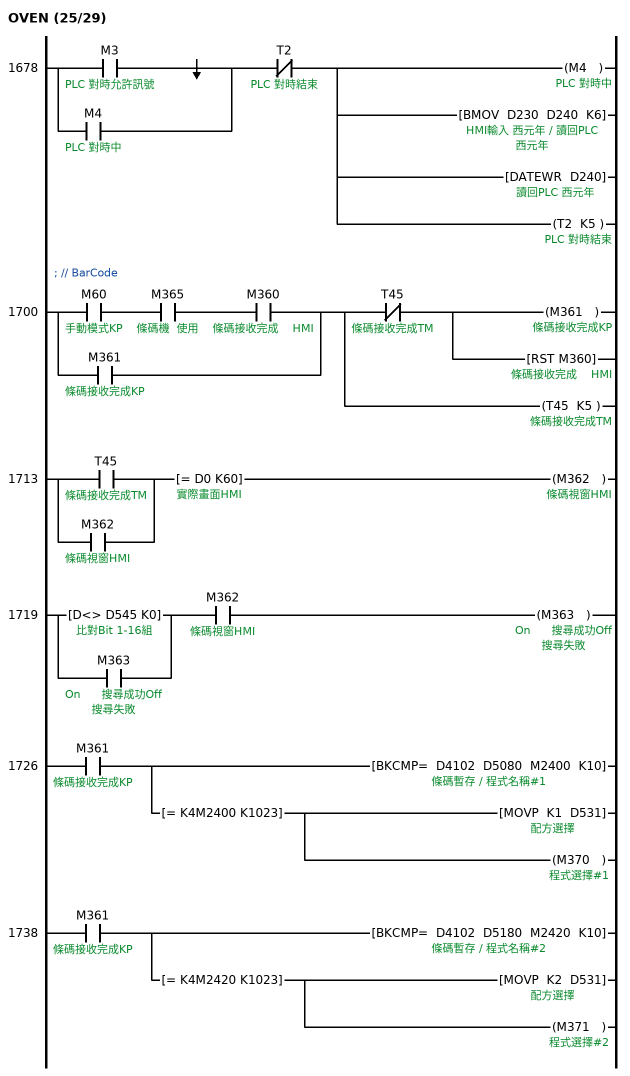
[picture p24: ladder of OVEN, rungs at steps 1678 to 1738]
1678  LD      M3  ; PLC 對時允許訊號
      MEF
      OR      M4  ; PLC 對時中
      ANI     T2  ; PLC 對時結束
      OUT     M4  ; PLC 對時中
      BMOV    D230 D240 K6
      DATEWR  D240
      OUT     T2 K5  ; PLC 對時結束
; // BarCode
1700  LD      M60  ; 手動模式KP
      AND     M365  ; 條碼機  使用
      AND     M360  ; 條碼接收完成    HMI
      OR      M361  ; 條碼接收完成KP
      MPS
      ANI     T45  ; 條碼接收完成TM
      OUT     M361  ; 條碼接收完成KP
      RST     M360  ; 條碼接收完成    HMI
      MPP
      OUT     T45 K5  ; 條碼接收完成TM
1713  LD      T45  ; 條碼接收完成TM
      OR      M362  ; 條碼視窗HMI
      AND=    D0 K60  ; 實際畫面HMI
      OUT     M362  ; 條碼視窗HMI
1719  LDD<>   D545 K0  ; 比對Bit 1-16組
      OR      M363  ; On      搜尋成功Off     搜尋失敗
      AND     M362  ; 條碼視窗HMI
      OUT     M363  ; On      搜尋成功Off     搜尋失敗
1726  LD      M361  ; 條碼接收完成KP
      BKCMP=  D4102 D5080 M2400 K10  ; 條碼暫存 / 程式名稱#1
      AND=    K4M2400 K1023
      MOVP    K1 D531
      OUT     M370  ; 程式選擇#1
1738  LD      M361  ; 條碼接收完成KP
      BKCMP=  D4102 D5180 M2420 K10  ; 程式名稱#2
      AND=    K4M2420 K1023
      MOVP    K2 D531
      OUT     M371  ; 程式選擇#2
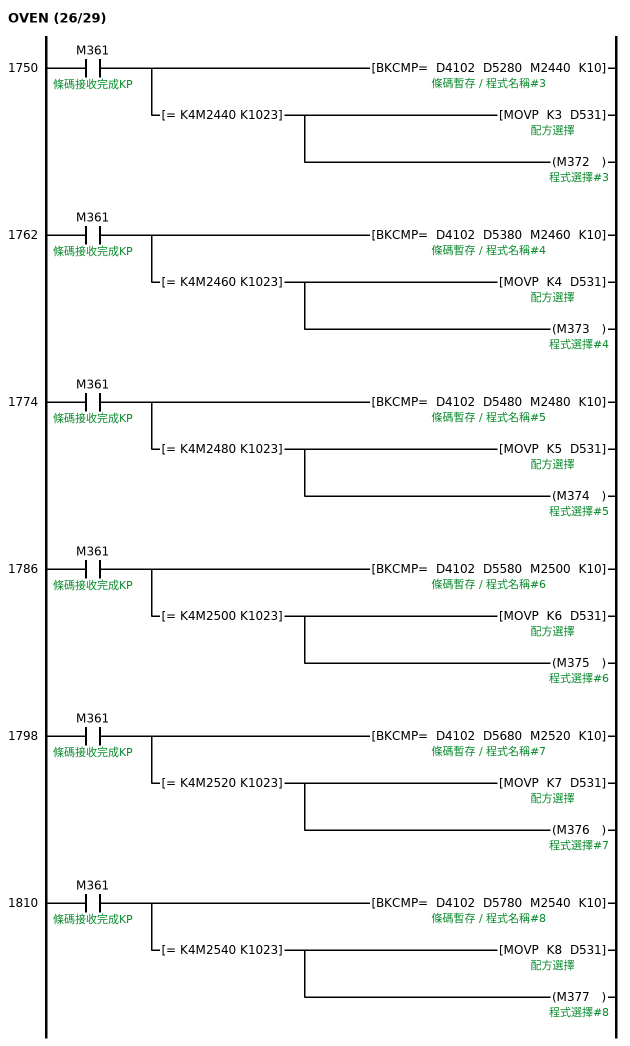
1750  LD      M361  ; 條碼接收完成KP
      BKCMP=  D4102 D5280 M2440 K10  ; 程式名稱#3
      AND=    K4M2440 K1023
      MOVP    K3 D531
      OUT     M372  ; 程式選擇#3
1762  LD      M361  ; 條碼接收完成KP
      BKCMP=  D4102 D5380 M2460 K10  ; 程式名稱#4
      AND=    K4M2460 K1023
      MOVP    K4 D531
      OUT     M373  ; 程式選擇#4
1774  LD      M361  ; 條碼接收完成KP
      BKCMP=  D4102 D5480 M2480 K10  ; 程式名稱#5
      AND=    K4M2480 K1023
      MOVP    K5 D531
      OUT     M374  ; 程式選擇#5
1786  LD      M361  ; 條碼接收完成KP
      BKCMP=  D4102 D5580 M2500 K10  ; 程式名稱#6
      AND=    K4M2500 K1023
      MOVP    K6 D531
      OUT     M375  ; 程式選擇#6
1798  LD      M361  ; 條碼接收完成KP
      BKCMP=  D4102 D5680 M2520 K10  ; 程式名稱#7
      AND=    K4M2520 K1023
      MOVP    K7 D531
      OUT     M376  ; 程式選擇#7
1810  LD      M361  ; 條碼接收完成KP
      BKCMP=  D4102 D5780 M2540 K10  ; 程式名稱#8
      AND=    K4M2540 K1023
      MOVP    K8 D531
      OUT     M377  ; 程式選擇#8
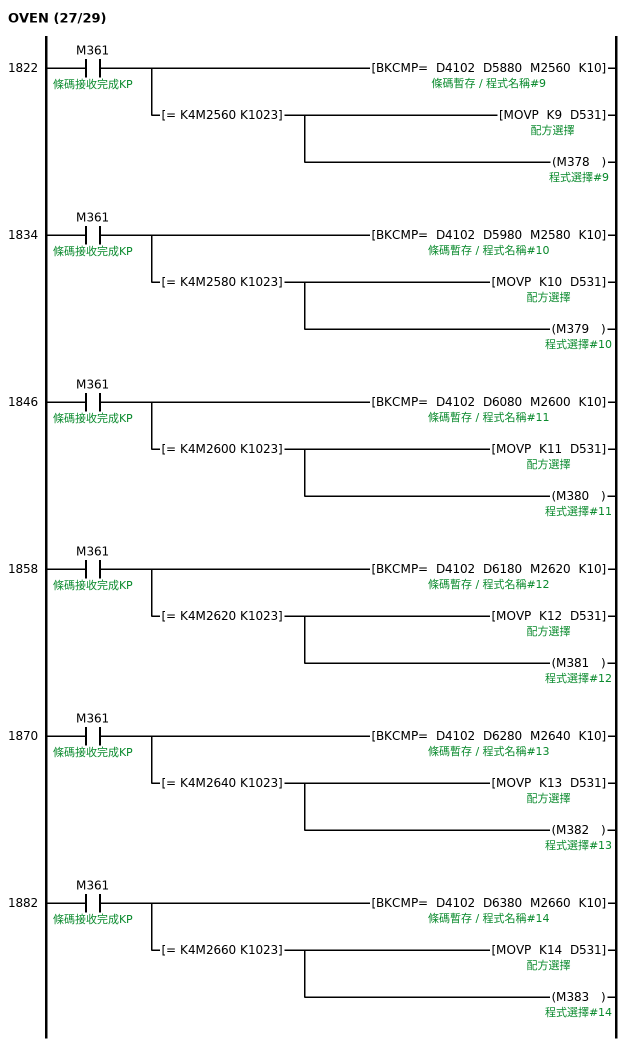
1822  LD      M361  ; 條碼接收完成KP
      BKCMP=  D4102 D5880 M2560 K10  ; 程式名稱#9
      AND=    K4M2560 K1023
      MOVP    K9 D531
      OUT     M378  ; 程式選擇#9
1834  LD      M361  ; 條碼接收完成KP
      BKCMP=  D4102 D5980 M2580 K10  ; 程式名稱#10
      AND=    K4M2580 K1023
      MOVP    K10 D531
      OUT     M379  ; 程式選擇#10
1846  LD      M361  ; 條碼接收完成KP
      BKCMP=  D4102 D6080 M2600 K10  ; 程式名稱#11
      AND=    K4M2600 K1023
      MOVP    K11 D531
      OUT     M380  ; 程式選擇#11
1858  LD      M361  ; 條碼接收完成KP
      BKCMP=  D4102 D6180 M2620 K10  ; 程式名稱#12
      AND=    K4M2620 K1023
      MOVP    K12 D531
      OUT     M381  ; 程式選擇#12
1870  LD      M361  ; 條碼接收完成KP
      BKCMP=  D4102 D6280 M2640 K10  ; 程式名稱#13
      AND=    K4M2640 K1023
      MOVP    K13 D531
      OUT     M382  ; 程式選擇#13
1882  LD      M361  ; 條碼接收完成KP
      BKCMP=  D4102 D6380 M2660 K10  ; 程式名稱#14
      AND=    K4M2660 K1023
      MOVP    K14 D531
      OUT     M383  ; 程式選擇#14
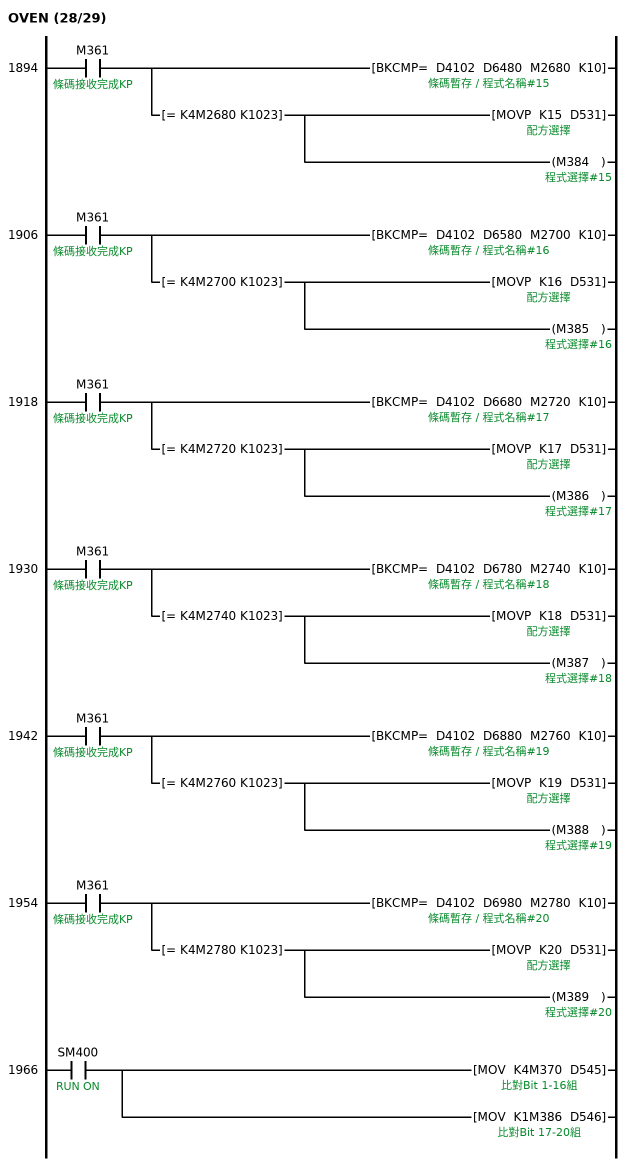
1894  LD      M361  ; 條碼接收完成KP
      BKCMP=  D4102 D6480 M2680 K10  ; 程式名稱#15
      AND=    K4M2680 K1023
      MOVP    K15 D531
      OUT     M384  ; 程式選擇#15
1906  LD      M361  ; 條碼接收完成KP
      BKCMP=  D4102 D6580 M2700 K10  ; 程式名稱#16
      AND=    K4M2700 K1023
      MOVP    K16 D531
      OUT     M385  ; 程式選擇#16
1918  LD      M361  ; 條碼接收完成KP
      BKCMP=  D4102 D6680 M2720 K10  ; 程式名稱#17
      AND=    K4M2720 K1023
      MOVP    K17 D531
      OUT     M386  ; 程式選擇#17
1930  LD      M361  ; 條碼接收完成KP
      BKCMP=  D4102 D6780 M2740 K10  ; 程式名稱#18
      AND=    K4M2740 K1023
      MOVP    K18 D531
      OUT     M387  ; 程式選擇#18
1942  LD      M361  ; 條碼接收完成KP
      BKCMP=  D4102 D6880 M2760 K10  ; 程式名稱#19
      AND=    K4M2760 K1023
      MOVP    K19 D531
      OUT     M388  ; 程式選擇#19
1954  LD      M361  ; 條碼接收完成KP
      BKCMP=  D4102 D6980 M2780 K10  ; 程式名稱#20
      AND=    K4M2780 K1023
      MOVP    K20 D531
      OUT     M389  ; 程式選擇#20
1966  LD      SM400  ; RUN ON
      MOV     K4M370 D545
      MOV     K1M386 D546  ; 比對Bit 17-20組
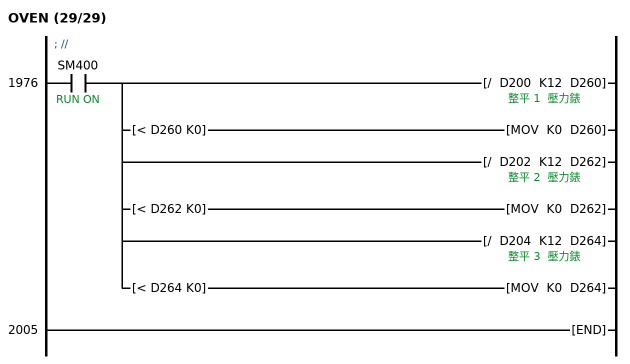
; //
1976  LD      SM400  ; RUN ON
      /       D200 K12 D260  ; 整平 1  壓力錶
      MPS
      AND<    D260 K0
      MOV     K0 D260
      MPP
      /       D202 K12 D262  ; 整平 2  壓力錶
      MPS
      AND<    D262 K0
      MOV     K0 D262
      MPP
      /       D204 K12 D264  ; 整平 3  壓力錶
      AND<    D264 K0
      MOV     K0 D264
2005  END
END_PROGRAM

PROGRAM SECS
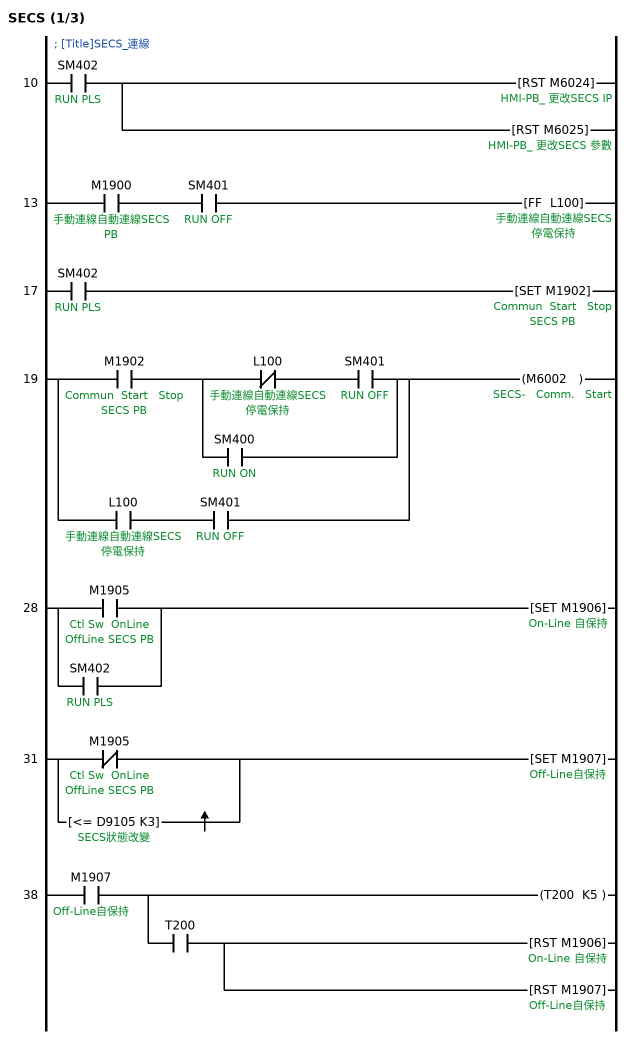
; [Title]SECS_連線
10    LD      SM402  ; RUN PLS
      RST     M6024  ; HMI-PB_ 更改SECS IP
      RST     M6025  ; HMI-PB_ 更改SECS 參數
13    LD      M1900  ; 手動連線自動連線SECS PB
      AND     SM401  ; RUN OFF
      FF      L100  ; 手動連線自動連線SECS    停電保持
17    LD      SM402  ; RUN PLS
      SET     M1902  ; Commun  Start   Stop    SECS PB
19    LD      M1902  ; Commun  Start   Stop    SECS PB
      LDI     L100  ; 手動連線自動連線SECS    停電保持
      AND     SM401  ; RUN OFF
      OR      SM400  ; RUN ON
      ANB
      LD      L100  ; 手動連線自動連線SECS    停電保持
      AND     SM401  ; RUN OFF
      ORB
      OUT     M6002  ; SECS-   Comm.   Start
28    LD      M1905  ; Ctl Sw  OnLine  OffLine SECS PB
      OR      SM402  ; RUN PLS
      SET     M1906  ; On-Line 自保持
31    LDI     M1905  ; Ctl Sw  OnLine  OffLine SECS PB
      LD<=    D9105 K3  ; SECS狀態改變
      MEP
      ORB
      SET     M1907  ; Off-Line自保持
38    LD      M1907  ; Off-Line自保持
      OUT     T200 K5
      AND     T200
      RST     M1906  ; On-Line 自保持
      RST     M1907  ; Off-Line自保持
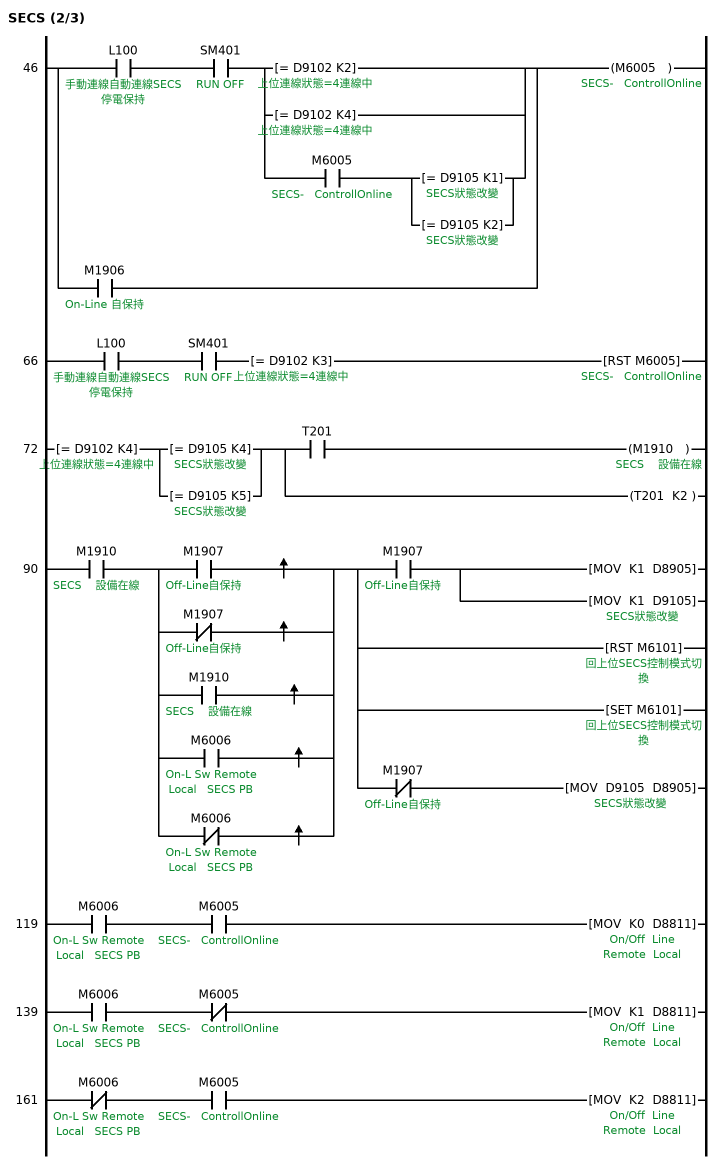
46    LD      L100  ; 手動連線自動連線SECS    停電保持
      AND     SM401  ; RUN OFF
      LD=     D9102 K2  ; 上位連線狀態=4連線中
      OR=     D9102 K4  ; 上位連線狀態=4連線中
      LD      M6005  ; SECS-   ControllOnline
      LD=     D9105 K1  ; SECS狀態改變
      OR=     D9105 K2  ; SECS狀態改變
      ANB
      ORB
      ANB
      OR      M1906  ; On-Line 自保持
      OUT     M6005  ; SECS-   ControllOnline
66    LD      L100  ; 手動連線自動連線SECS    停電保持
      AND     SM401  ; RUN OFF
      AND=    D9102 K3  ; 上位連線狀態=4連線中
      RST     M6005  ; SECS-   ControllOnline
72    LD=     D9102 K4  ; 上位連線狀態=4連線中
      LD=     D9105 K4  ; SECS狀態改變
      OR=     D9105 K5  ; SECS狀態改變
      ANB
      MPS
      AND     T201
      OUT     M1910  ; SECS    設備在線
      MPP
      OUT     T201 K2
90    LD      M1910  ; SECS    設備在線
      LD      M1907  ; Off-Line自保持
      MEP
      LDI     M1907  ; Off-Line自保持
      MEP
      ORB
      LD      M1910  ; SECS    設備在線
      MEP
      ORB
      LD      M6006  ; On-L Sw Remote  Local   SECS PB
      MEP
      ORB
      LDI     M6006  ; On-L Sw Remote  Local   SECS PB
      MEP
      ORB
      ANB
      MPS
      AND     M1907  ; Off-Line自保持
      MOV     K1 D8905
      MOV     K1 D9105
      MPP
      RST     M6101  ; 回上位SECS控制模式切換
      SET     M6101  ; 回上位SECS控制模式切換
      ANI     M1907  ; Off-Line自保持
      MOV     D9105 D8905
119   LD      M6006  ; On-L Sw Remote  Local   SECS PB
      AND     M6005  ; SECS-   ControllOnline
      MOV     K0 D8811  ; On/Off  Line    Remote  Local
        [note] D8811=K0(遠程控制+SEC在線中)
139   LD      M6006  ; On-L Sw Remote  Local   SECS PB
      ANI     M6005  ; SECS-   ControllOnline
      MOV     K1 D8811
        [note] D8811= k1(遠程控制中+SEC離線中)
161   LDI     M6006  ; On-L Sw Remote  Local   SECS PB
      AND     M6005  ; SECS-   ControllOnline
      MOV     K2 D8811
        [note] D881=k2(遠程控制離線+SEC在線中)
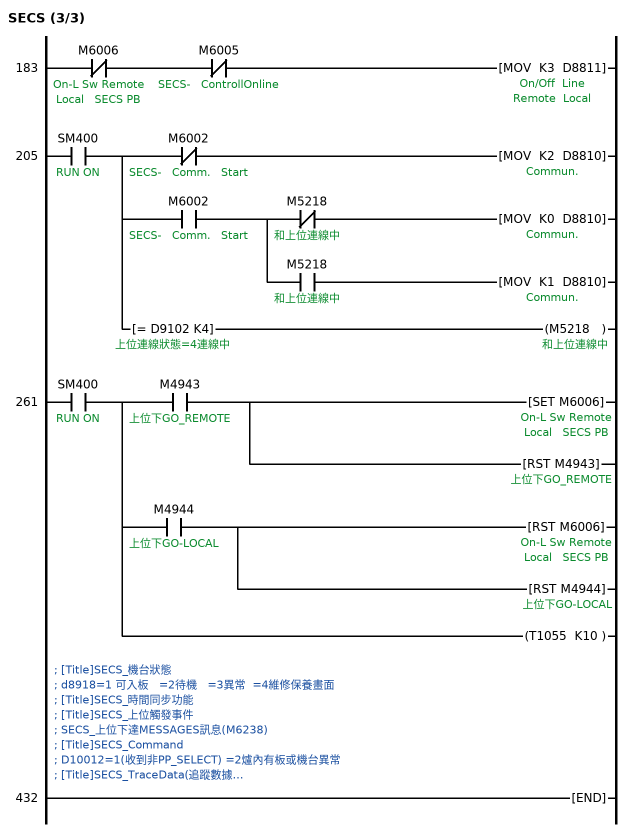
183   LDI     M6006  ; On-L Sw Remote  Local   SECS PB
      ANI     M6005  ; SECS-   ControllOnline
      MOV     K3 D8811
        [note] D881=k3(遠程控制離線+SEC離線中)
205   LD      SM400  ; RUN ON
      MPS
      ANI     M6002  ; SECS-   Comm.   Start
      MOV     K2 D8810  ; Commun.
        [note] K2= SEC通訊未連線
      MRD
      AND     M6002  ; SECS-   Comm.   Start
      MPS
      ANI     M5218  ; 和上位連線中
      MOV     K0 D8810
        [note] K0=SEC連線---上位未連線
      MPP
      AND     M5218  ; 和上位連線中
      MOV     K1 D8810
        [note] K1=SEC和上位連線中
      MPP
      AND=    D9102 K4  ; 上位連線狀態=4連線中
      OUT     M5218  ; 和上位連線中
261   LD      SM400  ; RUN ON
      MPS
      AND     M4943  ; 上位下GO_REMOTE
      SET     M6006  ; On-L Sw Remote  Local   SECS PB
      RST     M4943  ; 上位下GO_REMOTE
      MRD
      AND     M4944  ; 上位下GO-LOCAL
      RST     M6006  ; On-L Sw Remote  Local   SECS PB
      RST     M4944  ; 上位下GO-LOCAL
      MPP
      OUT     T1055 K10
; [Title]SECS_機台狀態
; d8918=1 可入板   =2待機   =3異常  =4維修保養畫面
; [Title]SECS_時間同步功能
; [Title]SECS_上位觸發事件
; SECS_上位下達MESSAGES訊息(M6238)
; [Title]SECS_Command
; D10012=1(收到非PP_SELECT) =2爐內有板或機台異常
; [Title]SECS_TraceData(追蹤數據)
; SECS_ALARM
; [Title]RECIPE_EDIT
432   END
END_PROGRAM

PROGRAM QJ71C24N
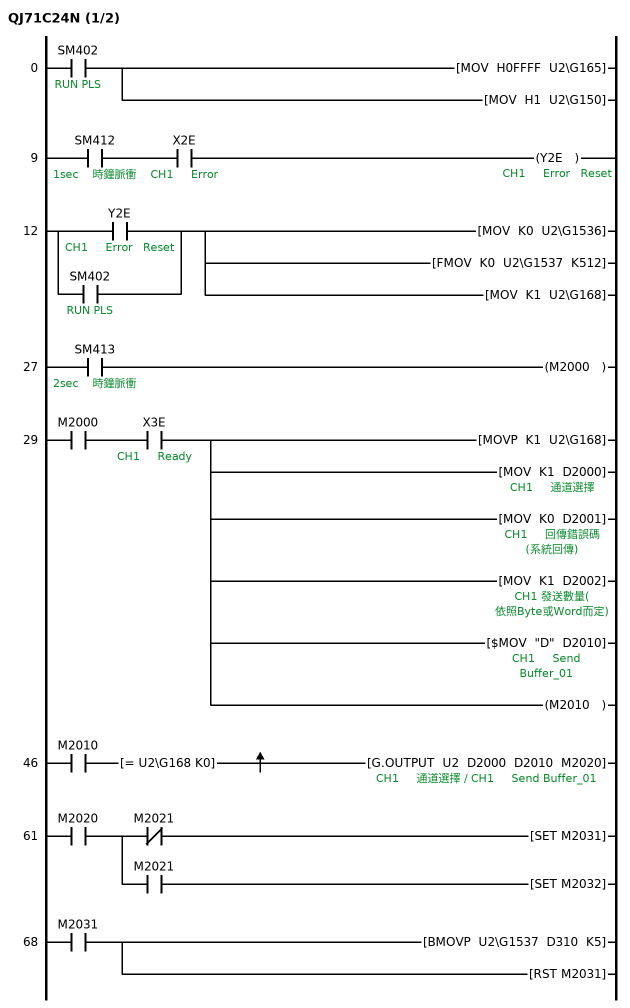
0     LD      SM402  ; RUN PLS
      MOV     H0FFFF U2\G165
      MOV     H1 U2\G150
9     LD      SM412  ; 1sec    時鐘脈衝
      AND     X2E  ; CH1     Error
      OUT     Y2E  ; CH1     Error   Reset
12    LD      Y2E  ; CH1     Error   Reset
      OR      SM402  ; RUN PLS
      MOV     K0 U2\G1536
      FMOV    K0 U2\G1537 K512
      MOV     K1 U2\G168
27    LD      SM413  ; 2sec    時鐘脈衝
      OUT     M2000
29    LD      M2000
      AND     X3E  ; CH1     Ready
      MOVP    K1 U2\G168
      MOV     K1 D2000  ; CH1     通道選擇
      MOV     K0 D2001  ; CH1     回傳錯誤碼  (系統回傳)
      MOV     K1 D2002  ; CH1 發送數量(依照Byte或Word而定)
      $MOV    "D" D2010  ; CH1     Send Buffer_01
      OUT     M2010
46    LD      M2010
      AND=    U2\G168 K0
      MEP
      G.OUTPUT U2 D2000 D2010 M2020
61    LD      M2020
      MPS
      ANI     M2021
      SET     M2031
      MPP
      AND     M2021
      SET     M2032
68    LD      M2031
      BMOVP   U2\G1537 D310 K5
      RST     M2031
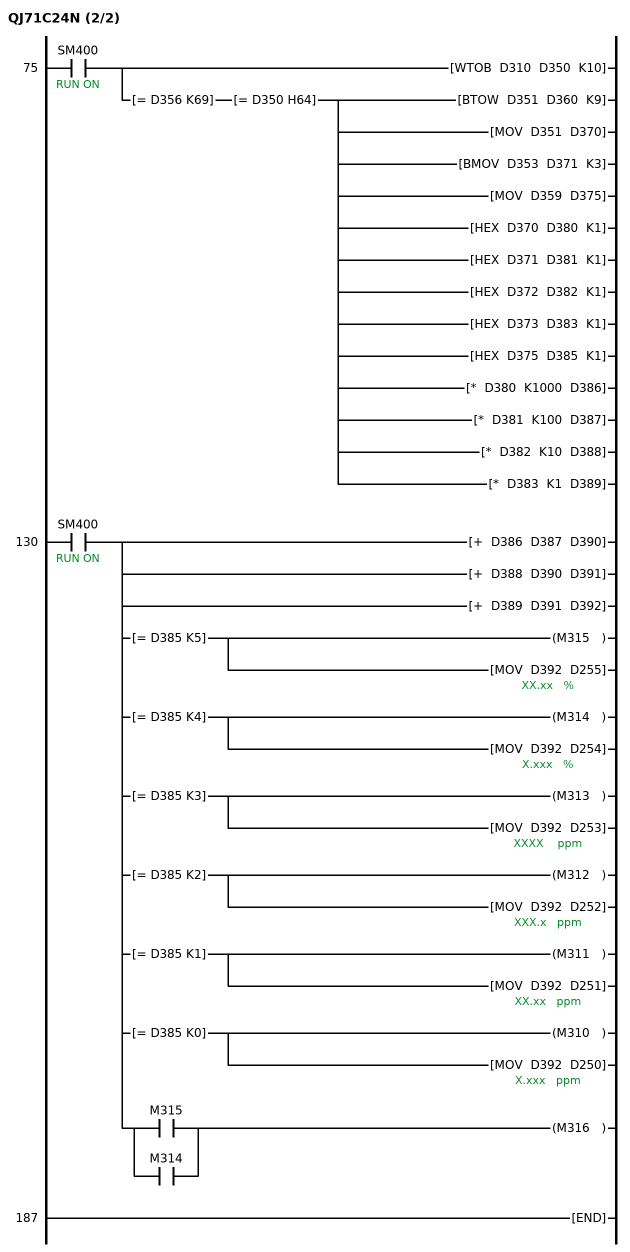
75    LD      SM400  ; RUN ON
      WTOB    D310 D350 K10
      AND=    D356 K69
      AND=    D350 H64
      BTOW    D351 D360 K9
      MOV     D351 D370
      BMOV    D353 D371 K3
      MOV     D359 D375
      HEX     D370 D380 K1
      HEX     D371 D381 K1
      HEX     D372 D382 K1
      HEX     D373 D383 K1
      HEX     D375 D385 K1
      *       D380 K1000 D386
      *       D381 K100 D387
      *       D382 K10 D388
      *       D383 K1 D389
130   LD      SM400  ; RUN ON
      +       D386 D387 D390
      +       D388 D390 D391
      +       D389 D391 D392
      MPS
      AND=    D385 K5
      OUT     M315
      MOV     D392 D255  ; XX.xx   %
      MRD
      AND=    D385 K4
      OUT     M314
      MOV     D392 D254  ; X.xxx   %
      MRD
      AND=    D385 K3
      OUT     M313
      MOV     D392 D253  ; XXXX    ppm
      MRD
      AND=    D385 K2
      OUT     M312
      MOV     D392 D252  ; XXX.x   ppm
      MRD
      AND=    D385 K1
      OUT     M311
      MOV     D392 D251  ; XX.xx   ppm
      MRD
      AND=    D385 K0
      OUT     M310
      MOV     D392 D250  ; X.xxx   ppm
      MPP
      LD      M315
      OR      M314
      ANB
      OUT     M316
187   END
END_PROGRAM

// device comments not shown above
M6238  ; 上位觸發開對話視窗
D810  ; 第01段  恆溫時間
D820  ; 第01段  升溫警報時間
D830  ; 第01段  恆溫警報時間
D840  ; 第01段  升溫時間
D855  ; 第01段  恆溫時間補償
D881  ; 程式名稱
D910  ; 第01段  恆溫+補償時間
D10012  ; 第03段  恆溫時間
M123  ; 電熱電磁開關LP
M133  ; 循環風車電磁開關LP
M138  ; 進氣風車電磁開關LP
M153  ; 排氣風門開啟繼電器LP
M163  ; 大量充氮氣繼電器LP
M168  ; 小量充氮氣繼電器LP
M1908  ; 對話視窗關閉 KP
M1920  ; 對話視窗打開 KP
M1921  ; 對話視窗關閉 PB
M3010  ; BC下發程式參數-執行
M3011  ; BC下發執行NG
M3012  ; BC下發執行-下載完成
M4000  ; BC下發參數名稱有效OK
M4001  ; BC下發參數名稱有效-1
M4002  ; BC下發參數名稱有效-2
M4003  ; BC下發參數機台不在自動啟動狀態
M4010  ; BC下發程式參數-執行\
M4011  ; BC下發執行NG
M4012  ; BC下發執行-下載完成
M4903  ; 爐內無板
M4920  ; 入口計數自保持
M4945  ; 上位允許放板START保持
M4946  ; 未達start 條件
M4948  ; 爐內片數=0
M4949  ; 機台自動生產中
M4950  ; 機台停止中(手動)
M4951  ; 上位允許切換配方自保持
M4952  ; S:切換配方動作流程切???
M4953  ; S:切換配方動作流程切啟動
M4954  ; S:手動狀態保持
M5204  ; 上位START-啟動
M5205  ; 上位STOP-停止
M5206  ; 上位允許切換配方
M5207  ; 上位切換成GO-REMOTE
M5208  ; 上位切換成GO-LOCAL
M5209  ; 上位下暫停進板
M5210  ; 上位下恢復進板
M5214  ; SECS上位下指令觸發Cmd-燈號
M5323  ; 緊急停止開關
M6009  ; 異常發生回報
M6010  ; 異常排除回報
M6014  ; 配方同步SET M6058
M6042  ; SECS上位下指令觸發Cmd
M6043  ; 通知SECS上位處理完畢(上位復歸)
M6050  ; SECS_LOG OUTPUT
M6052  ; PLC_LOG OUTPUT
M6058  ; 配方目錄同步R5300
M6059  ; Host刪除配方
M6060  ; Host刪除配方完成
M6102  ; 回上位機台狀態改變
M6103  ; 回上位自動啟動
M6104  ; 回上位當前使用配方變更
M6105  ; 回上位新增配方
M6106  ; 回上位刪除配方
M6107  ; 回上位修改配方
M6108  ; 回上位配方切換成功
M6109  ; 回上位Panel生產開始訊號
M6110  ; 回上位Panel生產結束訊號
M6111  ; 回上位Lot生產開始訊號
M6112  ; 回上位Lot生產結束訊號
M6113  ; 回上位配方狀態變更開始(開始升溫)
M6114  ; 回上位配方狀態變更結束(溫度到達)
M6115  ; PP_SELECT升溫中被中斷
M6116  ; SECS狀態改變中
M6117  ; 設備生產訊號收集-自動生產條件到
M6131  ; 生產完成程式結束
M6132  ; 機台狀態改變
M6134  ; 三色燈狀態改變
M6135  ; 回上位緊急停止開關訊號
M6136  ; 三色燈狀態改變
M6137  ; 手動
M6138  ; 確認讀取
M6140  ; 要求上位回讀工單板號右爐
M6141  ; 要求上位回讀工單右爐
M6142  ; 三色黃燈
M6218  ; 和上位連線中
M6233  ; 上位要配方內容
M6320  ; FX機台狀態改變
D8  ; 跳轉畫面HMI
D35  ; 升溫時間0.01 SEC
D37  ; 升溫每0.1℃間隔時間0.01 SEC
D38  ; 升溫每0.1℃間隔時間餘數
D39  ; 升溫每0.1℃間隔時間餘數
D96  ; J7800   (R)
D141  ; 第02段  升溫時間PV
D142  ; 第03段  升溫時間PV
D143  ; 第04段  升溫時間PV
D144  ; 第05段  升溫時間PV
D145  ; 第06段  升溫時間PV
D241  ; 讀回PLC月
D242  ; 讀回PLC日
D243  ; 讀回PLC時
D244  ; 讀回PLC分
D245  ; 讀回PLC秒
D400  ; EM330
D812  ; 第03段  恆溫時間
D821  ; 第02段  升溫警報時間
D822  ; 第03段  升溫警報時間
D823  ; 第04段  升溫警報時間
D824  ; 第05段  升溫警報時間
D825  ; 第06段  升溫警報時間
D841  ; 第02段  升溫時間
D842  ; 第03段  升溫時間
D843  ; 第04段  升溫時間
D844  ; 第05段  升溫時間
D845  ; 第06段  升溫時間
D854  ; Alarm reset timer
D911  ; 第02段  恆溫+補償時間
D912  ; 第03段  恆溫+補償時間
D913  ; 第04段  恆溫+補償時間
D914  ; 第05段  恆溫+補償時間
D915  ; 第06段  恆溫+補償時間
D7000  ; 第01段  目標溫度
D7010  ; 第01段  恆溫時間
D7012  ; 第03段  恆溫時間
D7020  ; 第01段  昇溫警報時間
D7021  ; 第02段  昇溫警報時間
D7022  ; 第03段  昇溫警報時間
D7023  ; 第04段  昇溫警報時間
D7024  ; 第05段  昇溫警報時間
D7025  ; 第06段  昇溫警報時間
D7030  ; 第01段  恆溫警報時間
D7040  ; 第01段  昇溫時間
D7041  ; 第02段  昇溫時間
D7042  ; 第03段  昇溫時間
D7043  ; 第04段  昇溫時間
D7044  ; 第05段  昇溫時間
D7045  ; 第06段  昇溫時間
D7050  ; 使用段數
D7051  ; 降溫時間SV
D7052  ; 降溫警報溫度SV
D7053  ; 降溫蜂鳴時間SV
D7054  ; 下發程式參數-各段升降溫功能選擇
D10000  ; 第01段  目標溫度
D10010  ; 第01段  恆溫時間
D10020  ; 第01段  昇溫警報時間
D10021  ; 第02段  昇溫警報時間
D10022  ; 第03段  昇溫警報時間
D10023  ; 第04段  昇溫警報時間
D10024  ; 第05段  昇溫警報時間
D10025  ; 第06段  昇溫警報時間
D10030  ; 第01段  恆溫警報時間
D10040  ; 第01段  昇溫時間
D10041  ; 第02段  昇溫時間
D10042  ; 第03段  昇溫時間
D10043  ; 第04段  昇溫時間
D10044  ; 第05段  昇溫時間
D10045  ; 第06段  昇溫時間
D10050  ; 使用段數
D10051  ; 降溫時間SV
D10052  ; 降溫警報溫度SV
D10053  ; 降溫蜂鳴時間SV
D10054  ; 下發程式參數-各段升降溫功能選擇
D11800  ; 第01段  目標溫度(NO.19)
D11801  ; 第02段  目標溫度(NO.19)
D11802  ; 第03段  目標溫度(NO.19)
D11803  ; 第04段  目標溫度(NO.19)
D11804  ; 第05段  目標溫度(NO.19)
D11805  ; 第06段  目標溫度(NO.19)
D11810  ; 第01段  恆溫時間(NO.19)
D11811  ; 第02段  恆溫時間(NO.19)
D11812  ; 第03段  恆溫時間(NO.19)
D11813  ; 第04段  恆溫時間(NO.19)
D11814  ; 第05段  恆溫時間(NO.19)
D11815  ; 第06段  恆溫時間(NO.19)
D11820  ; 第01段  昇溫警報時間(NO.19)
D11821  ; 第02段  昇溫警報時間(NO.19)
D11822  ; 第03段  昇溫警報時間(NO.19)
D11823  ; 第04段  昇溫警報時間(NO.19)
D11824  ; 第05段  昇溫警報時間(NO.19)
D11825  ; 第06段  昇溫警報時間(NO.19)
D11830  ; 第01段  恆溫警報時間(NO.19)
D11831  ; 第02段  恆溫警報時間(NO.19)
D11832  ; 第03段  恆溫警報時間(NO.19)
D11833  ; 第04段  恆溫警報時間(NO.19)
D11834  ; 第05段  恆溫警報時間(NO.19)
D11835  ; 第06段  恆溫警報時間(NO.19)
D11840  ; 第01段  昇溫時間(NO.19)
D11841  ; 第02段  昇溫時間(NO.19)
D11842  ; 第03段  昇溫時間(NO.19)
D11843  ; 第04段  昇溫時間(NO.19)
D11844  ; 第05段  昇溫時間(NO.19)
D11845  ; 第06段  昇溫時間(NO.19)
D11850  ; 使用段數(NO.19)
D11851  ; 降溫時間SV(NO.19)
D11852  ; 降溫警報溫度SV(NO.19)
D11853  ; 降溫蜂鳴時間SV(NO.19)
D11854  ; Alarm reset timer(NO.19)
D11900  ; 第01段  目標溫度(NO.20)
D11901  ; 第02段  目標溫度(NO.20)
D11902  ; 第03段  目標溫度(NO.20)
D11903  ; 第04段  目標溫度(NO.20)
D11904  ; 第05段  目標溫度(NO.20)
D11905  ; 第06段  目標溫度(NO.20)
D11910  ; 第01段  恆溫時間(NO.20)
D11911  ; 第02段  恆溫時間(NO.20)
D11912  ; 第03段  恆溫時間(NO.20)
D11913  ; 第04段  恆溫時間(NO.20)
D11914  ; 第05段  恆溫時間(NO.20)
D11915  ; 第06段  恆溫時間(NO.20)
D11920  ; 第01段  昇溫警報時間(NO.20)
D11921  ; 第02段  昇溫警報時間(NO.20)
D11922  ; 第03段  昇溫警報時間(NO.20)
D11923  ; 第04段  昇溫警報時間(NO.20)
D11924  ; 第05段  昇溫警報時間(NO.20)
D11925  ; 第06段  昇溫警報時間(NO.20)
D11930  ; 第01段  恆溫警報時間(NO.20)
D11931  ; 第02段  恆溫警報時間(NO.20)
D11932  ; 第03段  恆溫警報時間(NO.20)
D11933  ; 第04段  恆溫警報時間(NO.20)
D11934  ; 第05段  恆溫警報時間(NO.20)
D11935  ; 第06段  恆溫警報時間(NO.20)
D11940  ; 第01段  昇溫時間(NO.20)
D11941  ; 第02段  昇溫時間(NO.20)
D11942  ; 第03段  昇溫時間(NO.20)
D11943  ; 第04段  昇溫時間(NO.20)
D11944  ; 第05段  昇溫時間(NO.20)
D11945  ; 第06段  昇溫時間(NO.20)
D11950  ; 使用段數(NO.20)
D11951  ; 降溫時間SV(NO.20)
D11952  ; 降溫警報溫度SV(NO.20)
D11953  ; 降溫蜂鳴時間SV(NO.20)
D11954  ; Alarm reset timer(NO.20)
C100  ; 升溫時間計時
C101  ; 恆溫時間計數
C102  ; 昇溫逾時計數
C106  ; 降溫時間計數
C107  ; 降溫警報時間
C108  ; 總烘烤  時間0.1M
C110  ; 溫度值  寫入2次
C111  ; 手動寫入Retry
C120  ; 單位時間
C121  ; Alarm reset timer
C130  ; 昇溫到達段數
C131  ; 恆溫到達段數
L54  ; 程式結束
L1019  ; 下爐測溫模式開啟中
L1020  ; 下爐有帳(判斷空框或有料用)
L1054  ; 程式結束
L1063  ; 下前有框光纖檢測(啟動)
L1064  ; 下後有框光纖檢測(啟動)
X23  ; CH1     Read    Request
